PROGRAM MAIN
VAR
END_VAR

END_PROGRAM

(* stored: Version 1.1.0.1
   POU MAIN: Id {40a81e7e-9eb3-43d1-8501-18158a7ada09} *)
